ABB RAPID module: 001A3CB2

MODULE Shape_3

    CONST robtarget Target_10:=[[500,749.9,0.146],[0,0.86623271,0.499640763,0],[0,0,0,0],[9E+09,9E+09,9E+09,9E+09,9E+09,9E+09]];
    CONST robtarget Target_20:=[[650,663.297459622,0.146],[0,0.866281002,0.499557029,0],[0,0,0,0],[9E+09,9E+09,9E+09,9E+09,9E+09,9E+09]];
    ![0,0.965,-0.259,0]


    PROC Shape_3_Move()

        MoveL Target_10,v1000,fine,AW_Gun\WObj:=Level_0;
        MoveL Target_20,v1000,fine,AW_Gun\WObj:=Level_0;

    ENDPROC

ENDMODULE
